(* IEC 61131-3 sources: std_i2980_v2.06_cp053/Source/IMM/ieccontrol/InjectionGeneral (part 3) *)

(* ---- ABBackPressureCalibCycle.pu ---- *)
(*
@h    ! WARNING !
@h    The Kemro K2 system (including software) only meets category B according to EN 954-1,
@h    thus it is not intended for usage in safety-relevant control applications in the field
@h    of personal safety (e.g. emergency stop).
@h    To implement potentially necessary safety-relevant control tasks, always use additional
@h    external safety devices that are intended for the particular purpose, and meet the necessary
@h    functional safety.
@h    For further information see EN 954-1 (EN ISO 13849-1) and/or the K2-x00 user manual, chapter
@h    "CE conformity, directives and standards".

Do steps for automatic hold pressure calibration
*)

IMPORT_OVER_LISTFILE
 SET_ALARM
, START_PROCESS_ALGORITHM
, cCompInjection
, cMoveFwd
, cMaxInjectionCount
, cMoveInjectCalib
, FBCheckReady
, tsDeviceId
, tevStartRequest
, tnOperationMode
, FBStopStartedMovements
, tsCalibMovement
, tsCalculatedInjectData2
, ABAutoCalibRedoListener
, tsControlParameters
, tsDeadTimeParameters
, tevStartRequestData
, tsCalculatedInjectData
, tyCalculatedDataArray
, tnCalibMode
, FBAutoCalibLog
, tsCalibShiftData
, KMEM_CreateData
, KMEM_Status

END_IMPORT

ALGORITHM_BLOCK ABBackPressureCalibCycle #DUMMY_EDIT_BLOCK

SYSTEM_VAR
 sv_OperationMode : tnOperationMode;
 sv_DeviceId : tsDeviceId;
 sv_CalibStateBackPressure : tsCalibMovement;
 sv_TmpInjectionData : tsCalculatedInjectData2;
 sv_bDoBackPressureCalib : BOOL;
 sv_HoldingControlParams : tsControlParameters;
 sv_HoldingDeadTimeParams : tsDeadTimeParameters;
END_VAR

SYSTEM_OBJECT
 TaskMid : TASK;
 evStartRequest : tevStartRequest;
 PU_Task_7 : TASK;
END_OBJECT

VAR
 fbCheckReady : FBCheckReady;
 InjDeviceId : tsDeviceId;
 fbStopStartedMovements : FBStopStartedMovements;
 abAutoCalibRedoListenerBackP : ABAutoCalibRedoListener;
END_VAR

PROCESS_ALGORITHM paRun ON TaskMid

VAR_TEMP
 tmpMeanData : tsCalculatedInjectData;
 i : DINT;
END_VAR

VAR
 evStartRequestData : tevStartRequestData;
 iInjectionCount : DINT;
 calculatedParameters : tyCalculatedDataArray;
 calibMode : tnCalibMode := tnCalibMode_Raising;
 fbLog : FBAutoCalibLog;
 ShiftData : tsCalibShiftData;
 ShiftArrayCreateData : KMEM_CreateData;
 MeasuredPresArrayCreateData : KMEM_CreateData;
 MeasuredOutputArrayCreateData : KMEM_CreateData;
 ThirdStageArrayCreateData : KMEM_CreateData;
 s : KMEM_Status;
 iSize : UDINT;
 rTmp : REAL;
END_VAR

(* IecGraph-Code *)

(* init step *)
INITIAL_STEP S_INIT:
AInit (P);
ACreateArrays (P);
END_STEP

ACTION AInit: #BEGIN_EDIT_BLOCK
InjDeviceId := sv_DeviceId;
sv_bDoBackPressureCalib := TRUE;
iInjectionCount := 1;
sv_TmpInjectionData.CalibMode := calibMode;
sv_TmpInjectionData.bValid := FALSE;

;#END_EDIT_BLOCK END_ACTION (*AInit*)

(* steps *)
STEP S_RESET:
AStopmovements (P);
Action24 (P);
END_STEP

ACTION Action24: #BEGIN_EDIT_BLOCK
IF sv_CalibStateBackPressure.Status <> tnCalibState_Error THEN
   sv_CalibStateBackPressure.Status := tnCalibState_Aborted;
   fbLog('Back pressure calib aborted');
ELSE
    fbLog('Back pressure calib error');
END_IF;

;#END_EDIT_BLOCK END_ACTION (*Action24*)
STEP S_STOP:
ADeleteArrays (P);
Action22 (P);
END_STEP

ACTION Action22: #BEGIN_EDIT_BLOCK
sv_bDoBackPressureCalib := FALSE;
STOP_PROCESS_ALGORITHM();

;#END_EDIT_BLOCK END_ACTION (*Action22*)
STEP S_INJECT:
ADoProfile (P);
Action9 (N);
END_STEP

ACTION Action9: #BEGIN_EDIT_BLOCK
fbCheckReady(DeviceId := InjDeviceId)

;#END_EDIT_BLOCK END_ACTION (*Action9*)
STEP S_WAIT_CALC:
END_STEP

STEP S_SAVE_CALC:
Action17 (P);
END_STEP

ACTION Action17: #BEGIN_EDIT_BLOCK
calculatedParameters[iInjectionCount] := sv_TmpInjectionData;

;#END_EDIT_BLOCK END_ACTION (*Action17*)
STEP S_NEXT_CYCLE:
Action16 (P);
END_STEP

ACTION Action16: #BEGIN_EDIT_BLOCK
iInjectionCount := iInjectionCount +1;

;#END_EDIT_BLOCK END_ACTION (*Action16*)
STEP S_DONE:
Action18 (P);
Action14 (P);
END_STEP

ACTION Action18: #BEGIN_EDIT_BLOCK
tmpMeanData.rControllerKR := 0.0;
tmpMeanData.rControllerW  := 0.0;
tmpMeanData.tPlantDeadTime:= t#0ms;
tmpMeanData.rPlantK       := 0.0;
tmpMeanData.tPlantT1      := t#0ms;
(* calculate mean value of all parameters *)
(* fixme: check if we need to calculate from falling and raising first
   and then calculate over the arry *)
FOR i:= 1 TO cMaxInjectionCount DO
    IF calibMode = tnCalibMode_Both THEN
        tmpMeanData.rControllerKR := tmpMeanData.rControllerKR + calculatedParameters[i].Falling.rControllerKR + calculatedParameters[i].Raising.rControllerKR;
        tmpMeanData.rControllerW  := tmpMeanData.rControllerW  + calculatedParameters[i].Falling.rControllerW  + calculatedParameters[i].Raising.rControllerW;
        tmpMeanData.tControllerTN := tmpMeanData.tControllerTN + calculatedParameters[i].Falling.tControllerTN + calculatedParameters[i].Raising.tControllerTN;
        tmpMeanData.tPlantDeadTime:= tmpMeanData.tPlantDeadTime+ calculatedParameters[i].Falling.tPlantDeadTime+ calculatedParameters[i].Raising.tPlantDeadTime;
        tmpMeanData.rPlantK       := tmpMeanData.rPlantK       + calculatedParameters[i].Falling.rPlantK       + calculatedParameters[i].Raising.rPlantK;
        tmpMeanData.tPlantT1      := tmpMeanData.tPlantT1      + calculatedParameters[i].Falling.tPlantT1      + calculatedParameters[i].Raising.tPlantT1;
       ELSIF calibMode = tnCalibMode_Raising THEN
        tmpMeanData.rControllerKR := tmpMeanData.rControllerKR + calculatedParameters[i].Raising.rControllerKR;
        tmpMeanData.rControllerW  := tmpMeanData.rControllerW  + calculatedParameters[i].Raising.rControllerW;
        tmpMeanData.tControllerTN := tmpMeanData.tControllerTN + calculatedParameters[i].Raising.tControllerTN;
        tmpMeanData.tPlantDeadTime:= tmpMeanData.tPlantDeadTime+ calculatedParameters[i].Raising.tPlantDeadTime;
        tmpMeanData.rPlantK       := tmpMeanData.rPlantK       + calculatedParameters[i].Raising.rPlantK;
        tmpMeanData.tPlantT1      := tmpMeanData.tPlantT1      + calculatedParameters[i].Raising.tPlantT1;
       ELSIF calibMode = tnCalibMode_Falling THEN
        tmpMeanData.rControllerKR := tmpMeanData.rControllerKR + calculatedParameters[i].Falling.rControllerKR ;
        tmpMeanData.rControllerW  := tmpMeanData.rControllerW  + calculatedParameters[i].Falling.rControllerW;
        tmpMeanData.tControllerTN := tmpMeanData.tControllerTN + calculatedParameters[i].Falling.tControllerTN;
        tmpMeanData.tPlantDeadTime:= tmpMeanData.tPlantDeadTime+ calculatedParameters[i].Falling.tPlantDeadTime;
        tmpMeanData.rPlantK       := tmpMeanData.rPlantK       + calculatedParameters[i].Falling.rPlantK;
        tmpMeanData.tPlantT1      := tmpMeanData.tPlantT1      + calculatedParameters[i].Falling.tPlantT1;
    END_IF;
END_FOR;

tmpMeanData.rControllerKR := tmpMeanData.rControllerKR / DINT_TO_REAL(cMaxInjectionCount);
tmpMeanData.rControllerW  := tmpMeanData.rControllerW  / DINT_TO_REAL(cMaxInjectionCount);
tmpMeanData.tControllerTN := tmpMeanData.tControllerTN / DINT_TO_REAL(cMaxInjectionCount);
tmpMeanData.tPlantDeadTime:= tmpMeanData.tPlantDeadTime/ DINT_TO_REAL(cMaxInjectionCount);
tmpMeanData.rPlantK       := tmpMeanData.rPlantK       / DINT_TO_REAL(cMaxInjectionCount);
tmpMeanData.tPlantT1      := tmpMeanData.tPlantT1      / DINT_TO_REAL(cMaxInjectionCount);

IF calibMode = tnCalibMode_Both THEN
    (* if only one edge no division is needed *)
    tmpMeanData.rControllerKR := tmpMeanData.rControllerKR / 2.0;
    tmpMeanData.rControllerW  := tmpMeanData.rControllerW  / 2.0;
    tmpMeanData.tControllerTN := DIVTIME(tmpMeanData.tControllerTN, 2);
    tmpMeanData.tPlantDeadTime:= DIVTIME(tmpMeanData.tPlantDeadTime, 2);
    tmpMeanData.rPlantK       := tmpMeanData.rPlantK/ 2.0;
    tmpMeanData.tPlantT1      := DIVTIME(tmpMeanData.tPlantT1, 2);
END_IF;

sv_HoldingControlParams.bUsePIDControl := TRUE;
sv_HoldingControlParams.rKS := 1.0;
sv_HoldingControlParams.dTN := tmpMeanData.tControllerTN;
sv_HoldingControlParams.dTV := t#0s;
sv_HoldingControlParams.rP := tmpMeanData.rControllerKR;

sv_HoldingDeadTimeParams.bCompensationEnabled := TRUE;
sv_HoldingDeadTimeParams.dDeadTime := tmpMeanData.tPlantDeadTime;
sv_HoldingDeadTimeParams.dPT2T1 := tmpMeanData.tPlantT1;
sv_HoldingDeadTimeParams.rPT2K := tmpMeanData.rPlantK;

sv_HoldingControlParams.bUsePIDControl := TRUE;

;#END_EDIT_BLOCK END_ACTION (*Action18*)
ACTION Action14: #BEGIN_EDIT_BLOCK
sv_CalibStateBackPressure.Status := tnCalibState_Done;

;#END_EDIT_BLOCK END_ACTION (*Action14*)

(* transitions *)
GO_ON_TRANSITION Trans15 (* Trans15 *) FROM S_RESET TO S_STOP :=  #BEGIN_EDIT_BLOCK
TRUE
;#END_EDIT_BLOCK
END_TRANSITION

TRANSITION Trans18 (* Trans18 *) FROM S_STOP TO S_INIT :=  #BEGIN_EDIT_BLOCK
TRUE
;#END_EDIT_BLOCK
END_TRANSITION

TRANSITION Trans1 (* Trans1 *) FROM S_INIT TO S_INJECT :=  #BEGIN_EDIT_BLOCK
TRUE
;#END_EDIT_BLOCK
END_TRANSITION

TRANSITION Trans2 (* Trans2 *) FROM S_INJECT TO S_WAIT_CALC :=  #BEGIN_EDIT_BLOCK
fbCheckReady.bReady AND S_INJECT.T >= t#1s
;#END_EDIT_BLOCK
(*Comment :FIXME: delay because else we sometimes get a erDeviceActive on first movement*)
END_TRANSITION

TRANSITION Trans21 (* Trans21 *) FROM S_WAIT_CALC TO S_SAVE_CALC :=  #BEGIN_EDIT_BLOCK
sv_TmpInjectionData.bValid
;#END_EDIT_BLOCK
END_TRANSITION

TRANSITION Trans22 (* Trans22 *) FROM S_WAIT_CALC TO S_RESET :=  #BEGIN_EDIT_BLOCK
sv_TmpInjectionData.bInvalid
;#END_EDIT_BLOCK
END_TRANSITION

TRANSITION Trans10 (* Trans10 *) FROM S_SAVE_CALC TO S_DONE :=  #BEGIN_EDIT_BLOCK
iInjectionCount >= cMaxInjectionCount
;#END_EDIT_BLOCK
END_TRANSITION

TRANSITION Trans11 (* Trans11 *) FROM S_SAVE_CALC TO S_NEXT_CYCLE :=  #BEGIN_EDIT_BLOCK
iInjectionCount < cMaxInjectionCount
;#END_EDIT_BLOCK
END_TRANSITION

TRANSITION Trans14 (* Trans14 *) FROM S_NEXT_CYCLE TO S_INJECT :=  #BEGIN_EDIT_BLOCK
TRUE
;#END_EDIT_BLOCK
END_TRANSITION

TRANSITION Trans19 (* Trans19 *) FROM S_DONE TO S_STOP :=  #BEGIN_EDIT_BLOCK
TRUE
;#END_EDIT_BLOCK
END_TRANSITION

(* end IecGraph-Code *)
(* sfc-code *)

(* stand alone actions *)
ACTION ADoProfile: #BEGIN_EDIT_BLOCK
evStartRequestData.DeviceId := InjDeviceId;
evStartRequestData.MoveDir := cMoveFwd;
evStartRequestData.MoveId := cMoveInjectCalib;
SET_EVENT(evStartRequest, evStartRequestData);

;#END_EDIT_BLOCK END_ACTION (*ADoProfile*)
ACTION AStopmovements: #BEGIN_EDIT_BLOCK
fbStopStartedMovements();

;#END_EDIT_BLOCK END_ACTION (*AStopmovements*)
ACTION ACreateArrays: #BEGIN_EDIT_BLOCK
(**************************************** WARNING ********************************************
 *** The KEBA Kemro K2 System including software is not intended for safety control tasks! ***
 ***                       For further information see Comment tab!                        ***
 *********************************************************************************************)

//create dynamic arrays which are necessary for PID parameter detection
iSize := DINT_TO_UDINT(cMaxShiftData) + 1;
ShiftArrayCreateData := KMEM_ArrayCreate(cCalibShiftData, ShiftData, iSize);

iSize := DINT_TO_UDINT(cMaxRecordedData);
MeasuredPresArrayCreateData := KMEM_ArrayCreate(cCalibMeasuredPres, rTmp, iSize);
MeasuredOutputArrayCreateData := KMEM_ArrayCreate(cCalibMeasuredOutput, rTmp, iSize);
ThirdStageArrayCreateData := KMEM_ArrayCreate(cCalibThirdStage, rTmp, iSize);

;#END_EDIT_BLOCK END_ACTION (*ACreateArrays*)
ACTION ADeleteArrays: #BEGIN_EDIT_BLOCK
(**************************************** WARNING ********************************************
 *** The KEBA Kemro K2 System including software is not intended for safety control tasks! ***
 ***                       For further information see Comment tab!                        ***
 *********************************************************************************************)

s := KMEM_ArrayDelete(ShiftArrayCreateData.Handle);
s := KMEM_ArrayDelete(MeasuredPresArrayCreateData.Handle);
s := KMEM_ArrayDelete(MeasuredOutputArrayCreateData.Handle);
s := KMEM_ArrayDelete(ThirdStageArrayCreateData.Handle);

;#END_EDIT_BLOCK END_ACTION (*ADeleteArrays*)

(* exits *)

EXIT_TRANSITION E_NotSetupMode := #BEGIN_EDIT_BLOCK
(**************************************** WARNING ********************************************
 *** The KEBA Kemro K2 System including software is not intended for safety control tasks! ***
 ***                       For further information see Comment tab!                        ***
 *********************************************************************************************)

sv_OperationMode <> nSetup
;#END_EDIT_BLOCK
PRIORITY 1 WITH  INITIAL_STEP S_RESET: END_STEP
END_TRANSITION

EXIT_TRANSITION E_NotCalibratingAnymore := #BEGIN_EDIT_BLOCK
// abort calibration, when not in running state and not finished
sv_CalibStateBackPressure.Status <> tnCalibState_Running AND (S_INIT.X (*OR S_FORWARD.X*) OR S_INJECT.X OR S_WAIT_CALC.X)
;#END_EDIT_BLOCK
PRIORITY 1 WITH  INITIAL_STEP S_RESET: END_STEP
END_TRANSITION
(* end sfc-code *)

END_ALGORITHM

POSTUPDATE_ALGORITHM pStart ON PU_Task_7 WITH sv_CalibStateBackPressure.Status

#BEGIN_EDIT_BLOCK
(**************************************** WARNING ********************************************
 *** The KEBA Kemro K2 System including software is not intended for safety control tasks! ***
 ***                       For further information see Comment tab!                        ***
 *********************************************************************************************)

IF sv_OperationMode = nSetup THEN
   IF sv_CalibStateBackPressure.Status = tnCalibState_Running THEN
      START_PROCESS_ALGORITHM(paRun);
   END_IF;
END_IF;

;#END_EDIT_BLOCK END_ALGORITHM

END_ALGORITHM_BLOCK

#END_OF_IEC_PART

@Puma @IecEditor 6 97 @Pou 25
@@@BEG_Comment@@@
@h    ! WARNING !
@h    The Kemro K2 system (including software) only meets category B according to EN 954-1,
@h    thus it is not intended for usage in safety-relevant control applications in the field
@h    of personal safety (e.g. emergency stop).
@h    To implement potentially necessary safety-relevant control tasks, always use additional
@h    external safety devices that are intended for the particular purpose, and meet the necessary
@h    functional safety.
@h    For further information see EN 954-1 (EN ISO 13849-1) and/or the K2-x00 user manual, chapter
@h    "CE conformity, directives and standards".

Do steps for automatic hold pressure calibration
@@@END_Comment@@@

@BEG_Contents

@BEG_Func
@RT(17)FuncTreeContainer
2
@Var @RT(9)SET_ALARM @RT(0) @T @T @DERIVED 0 @F @RT(23)KEBA_STANDARD_PROCEDURE @F
@T
@BEG_Attrib
0 @RT(0) @RT(0)
@END_Attrib
1 1 @F @F @F @F

@Var @RT(23)START_PROCESS_ALGORITHM @RT(0) @T @T @DERIVED 0 @F @RT(23)KEBA_STANDARD_PROCEDURE @F
@T
@BEG_Attrib
0 @RT(0) @RT(0)
@END_Attrib
1 1 @F @F @F @F

@END_Func

@BEG_Const
@RT(18)ConstTreeContainer
4
@Var @RT(14)cCompInjection @RT(0) @T @F @DT @RT(4)DINT @RT(0) @T @T @BASIC 0 @F
@F @F
@T
@BEG_Attrib
0 @RT(3)104 @RT(19)Component Injection
@END_Attrib
1 1 @F @F @F @F

@Var @RT(8)cMoveFwd @RT(0) @T @F @DT @RT(4)DINT @RT(0) @T @T @BASIC 0 @F
@F @F
@T
@BEG_Attrib
0 @RT(2)12 @RT(16)movement forward
@END_Attrib
1 1 @F @F @F @F

@Var @RT(18)cMaxInjectionCount @RT(0) @T @F @DT @RT(4)DINT @RT(0) @T @T @BASIC 0 @F
@F @F
@T
@BEG_Attrib
0 @RT(1)3 @RT(41)how often to do injection for calibration
@END_Attrib
1 1 @F @F @F @F

@Var @RT(16)cMoveInjectCalib @RT(0) @T @F @DT @RT(4)DINT @RT(0) @T @T @BASIC 0 @F
@F @F
@T
@BEG_Attrib
0 @RT(2)70 @RT(48)calibration movement for servo inject controller
@END_Attrib
1 1 @F @F @F @F

@END_Const

@BEG_Export

@BEG_Kind
@ALGORITHM_BLOCK @RT(24)ABBackPressureCalibCycle @STRUCTURED_TEXT
@RT(0) @RT(0) @RT(0)
@END_Kind

@BEG_Dcl
@RT(16)DclTreeContainer
14
@Var @RT(7)TaskMid @RT(0) @T @T @RENAMED 0 @T @T @DT @RT(4)TASK @RT(0) @T @T @BASIC 0 @F
@F @F
@T
@BEG_Attrib
3 @RT(0) @RT(0) @RT(0)
@END_Attrib
1 7 @F @F @F @F

@Var @RT(12)fbCheckReady @RT(0) @T @T @DERIVED 0 @T @T @DT @RT(12)FBCheckReady @RT(0) @T @T @UNKNOWN 0 @F
@F @F
@T
@BEG_Attrib
3 @RT(0) @RT(0) @RT(0)
@END_Attrib
1 0 @F @F @F @F

@Var @RT(11)InjDeviceId @RT(0) @T @T @DERIVED 0 @T @T @DT @RT(10)tsDeviceId @RT(0) @T @T @UNKNOWN 0 @F
@F @F
@T
@BEG_Attrib
3 @RT(0) @RT(0) @RT(0)
@END_Attrib
1 0 @F @F @F @F

@Var @RT(14)evStartRequest @RT(0) @T @T @DERIVED 0 @T @T @DT @RT(15)tevStartRequest @RT(0) @T @T @UNKNOWN 0 @F
@F @F
@T
@BEG_Attrib
3 @RT(0) @RT(0) @RT(0)
@END_Attrib
1 7 @F @F @F @F

@Var @RT(9)PU_Task_7 @RT(0) @T @T @RENAMED 0 @T @T @DT @RT(4)TASK @RT(0) @T @T @BASIC 0 @F
@F @F
@T
@BEG_Attrib
3 @RT(0) @RT(0) @RT(0)
@END_Attrib
1 7 @F @F @F @F

@Var @RT(16)sv_OperationMode @RT(0) @T @T @DERIVED 0 @T @T @DT @RT(15)tnOperationMode @RT(0) @T @T @UNKNOWN 0 @F
@F @F
@T
@BEG_Attrib
3 @RT(0) @RT(0) @RT(0)
@END_Attrib
1 8 @F @F @F @F

@Var @RT(22)fbStopStartedMovements @RT(0) @T @T @DERIVED 0 @T @T @DT @RT(22)FBStopStartedMovements @RT(0) @T @T @UNKNOWN 0 @F
@F @F
@T
@BEG_Attrib
3 @RT(0) @RT(0) @RT(0)
@END_Attrib
1 0 @F @F @F @F

@Var @RT(11)sv_DeviceId @RT(0) @T @T @RENAMED 0 @T @T @DT @RT(10)tsDeviceId @RT(0) @T @T @UNKNOWN 0 @F
@F @F
@T
@BEG_Attrib
3 @RT(0) @RT(0) @RT(0)
@END_Attrib
1 8 @F @F @F @F

@Var @RT(25)sv_CalibStateBackPressure @RT(0) @T @T @RENAMED 0 @T @T @DT @RT(15)tsCalibMovement @RT(0) @T @T @UNKNOWN 0 @F
@F @F
@T
@BEG_Attrib
3 @RT(0) @RT(0) @RT(0)
@END_Attrib
1 8 @F @F @F @F

@Var @RT(19)sv_TmpInjectionData @RT(0) @T @T @DERIVED 0 @T @T @DT @RT(23)tsCalculatedInjectData2 @RT(0) @T @T @UNKNOWN 0 @F
@F @F
@T
@BEG_Attrib
3 @RT(0) @RT(0) @RT(0)
@END_Attrib
1 8 @F @F @F @F

@Var @RT(23)sv_bDoBackPressureCalib @RT(0) @T @T @RENAMED 0 @T @T @DT @RT(4)BOOL @RT(0) @T @T @BASIC 0 @F
@F @F
@T
@BEG_Attrib
3 @RT(0) @RT(0) @RT(0)
@END_Attrib
1 8 @F @F @F @F

@Var @RT(28)abAutoCalibRedoListenerBackP @RT(0) @T @T @DERIVED 0 @T @T @DT @RT(23)ABAutoCalibRedoListener @RT(0) @T @T @UNKNOWN 0 @F
@F @F
@T
@BEG_Attrib
3 @RT(0) @RT(0) @RT(0)
@END_Attrib
1 0 @F @F @F @F

@Var @RT(23)sv_HoldingControlParams @RT(0) @T @T @RENAMED 0 @T @T @DT @RT(19)tsControlParameters @RT(0) @T @T @UNKNOWN 0 @F
@F @F
@T
@BEG_Attrib
3 @RT(0) @RT(0) @RT(0)
@END_Attrib
1 8 @F @F @F @F

@Var @RT(24)sv_HoldingDeadTimeParams @RT(0) @T @T @RENAMED 0 @T @T @DT @RT(20)tsDeadTimeParameters @RT(0) @T @T @UNKNOWN 0 @F
@F @F
@T
@BEG_Attrib
3 @RT(0) @RT(0) @RT(0)
@END_Attrib
1 8 @F @F @F @F

@END_Dcl

@END_Export

@BEG_Body

2

@BEG_Export

@BEG_Algo
@PROCESS_ALGORITHM @RT(5)paRun @SEQUENTIAL_FLOW_CHART
@RT(0) @RT(0) @RT(7)TaskMid @F @F
@END_Algo

@BEG_Dcl
@RT(16)DclTreeContainer
15
@Var @RT(18)evStartRequestData @RT(0) @T @T @DERIVED 0 @T @T @DT @RT(19)tevStartRequestData @RT(0) @T @T @UNKNOWN 0 @F
@F @F
@T
@BEG_Attrib
3 @RT(0) @RT(0) @RT(0)
@END_Attrib
1 0 @F @F @F @F

@Var @RT(15)iInjectionCount @RT(0) @T @F @DT @RT(4)DINT @RT(0) @T @T @BASIC 0 @F
@F @F
@T
@BEG_Attrib
3 @RT(0) @RT(0) @RT(0)
@END_Attrib
1 0 @F @F @F @F

@Var @RT(11)tmpMeanData @RT(0) @T @T @DERIVED 0 @T @T @DT @RT(22)tsCalculatedInjectData @RT(0) @T @T @UNKNOWN 0 @F
@F @F
@T
@BEG_Attrib
3 @RT(0) @RT(0) @RT(0)
@END_Attrib
1 4 @F @F @F @F

@Var @RT(20)calculatedParameters @RT(0) @T @T @DERIVED 0 @T @T @DT @RT(21)tyCalculatedDataArray @RT(0) @T @T @UNKNOWN 0 @F
@F @F
@T
@BEG_Attrib
3 @RT(0) @RT(0) @RT(0)
@END_Attrib
1 0 @F @F @F @F

@Var @RT(1)i @RT(0) @T @F @DT @RT(4)DINT @RT(0) @T @T @BASIC 0 @F
@F @F
@T
@BEG_Attrib
3 @RT(0) @RT(0) @RT(0)
@END_Attrib
1 4 @F @F @F @F

@Var @RT(9)calibMode @RT(0) @T @T @DERIVED 0 @T @T @DT @RT(11)tnCalibMode @RT(0) @T @T @UNKNOWN 0 @F
@F @F
@T
@BEG_Attrib
3 @RT(19)tnCalibMode_Raising @RT(0) @RT(0)
@END_Attrib
1 0 @F @F @F @F

@Var @RT(5)fbLog @RT(0) @T @T @DERIVED 0 @T @T @DT @RT(14)FBAutoCalibLog @RT(0) @T @T @UNKNOWN 0 @F
@F @F
@T
@BEG_Attrib
3 @RT(0) @RT(0) @RT(0)
@END_Attrib
1 0 @F @F @F @F

@Var @RT(9)ShiftData @RT(0) @T @T @DERIVED 0 @T @T @DT @RT(16)tsCalibShiftData @RT(0) @T @T @UNKNOWN 0 @F
@F @F
@T
@BEG_Attrib
3 @RT(0) @RT(0) @RT(0)
@END_Attrib
1 0 @F @F @F @F

@Var @RT(20)ShiftArrayCreateData @RT(0) @T @T @DERIVED 0 @T @T @DT @RT(15)KMEM_CreateData @RT(0) @T @T @UNKNOWN 0 @F
@F @F
@T
@BEG_Attrib
3 @RT(0) @RT(0) @RT(0)
@END_Attrib
1 0 @F @F @F @F

@Var @RT(27)MeasuredPresArrayCreateData @RT(0) @T @T @DERIVED 0 @T @T @DT @RT(15)KMEM_CreateData @RT(0) @T @T @UNKNOWN 0 @F
@F @F
@T
@BEG_Attrib
3 @RT(0) @RT(0) @RT(0)
@END_Attrib
1 0 @F @F @F @F

@Var @RT(29)MeasuredOutputArrayCreateData @RT(0) @T @T @DERIVED 0 @T @T @DT @RT(15)KMEM_CreateData @RT(0) @T @T @UNKNOWN 0 @F
@F @F
@T
@BEG_Attrib
3 @RT(0) @RT(0) @RT(0)
@END_Attrib
1 0 @F @F @F @F

@Var @RT(25)ThirdStageArrayCreateData @RT(0) @T @T @DERIVED 0 @T @T @DT @RT(15)KMEM_CreateData @RT(0) @T @T @UNKNOWN 0 @F
@F @F
@T
@BEG_Attrib
3 @RT(0) @RT(0) @RT(0)
@END_Attrib
1 0 @F @F @F @F

@Var @RT(1)s @RT(0) @T @T @DERIVED 0 @T @T @DT @RT(11)KMEM_Status @RT(0) @T @T @UNKNOWN 0 @F
@F @F
@T
@BEG_Attrib
3 @RT(0) @RT(0) @RT(0)
@END_Attrib
1 0 @F @F @F @F

@Var @RT(5)iSize @RT(0) @T @F @DT @RT(5)UDINT @RT(0) @T @T @BASIC 0 @F
@F @F
@T
@BEG_Attrib
3 @RT(0) @RT(0) @RT(0)
@END_Attrib
1 0 @F @F @F @F

@Var @RT(4)rTmp @RT(0) @T @F @DT @RT(4)REAL @RT(0) @T @T @BASIC 0 @F
@F @F
@T
@BEG_Attrib
3 @RT(0) @RT(0) @RT(0)
@END_Attrib
1 0 @F @F @F @F

@END_Dcl

@END_Export

@BEG_Export

@BEG_Algo
@POSTUPDATE_ALGORITHM @RT(6)pStart @STRUCTURED_TEXT
@RT(0) @RT(32)sv_CalibStateBackPressure.Status @RT(9)PU_Task_7 @F @F
@END_Algo

@BEG_Dcl
@RT(16)DclTreeContainer
0
@END_Dcl

@END_Export

@BEG_SfcBody
26 17 23

@BEG_SfcData 2
@StepSeq @RT(4)sseq @F 15
@Step @RT(7)S_RESET @F @F @T @F @RT(0) @F
@AcbCont @RT(7)unnamed @F 2
@Acb @RT(14)AStopmovements @F @F @RT(1)P @RT(0) @F @F @T @F
@Acb @RT(8)Action24 @F @T @RT(1)P @RT(0) @F @F @T @TL(7)
IF sv_CalibStateBackPressure.Status <> tnCalibState_Error THEN
   sv_CalibStateBackPressure.Status := tnCalibState_Aborted;
   fbLog('Back pressure calib aborted');
ELSE
    fbLog('Back pressure calib error');
END_IF;

@F

@Trans @RT(7)Trans15 @F @T @F @F @T @F @TL(2)
TRUE

@RT(7)Trans15 @F
@Step @RT(6)S_STOP @F @F @T @F @RT(0) @F
@AcbCont @RT(7)unnamed @F 2
@Acb @RT(13)ADeleteArrays @F @F @RT(1)P @RT(0) @F @F @F @F
@Acb @RT(8)Action22 @F @T @RT(1)P @RT(0) @F @F @T @TL(3)
sv_bDoBackPressureCalib := FALSE;
STOP_PROCESS_ALGORITHM();

@F

@Trans @RT(7)Trans18 @F @T @F @F @T @T @TL(2)
TRUE

@RT(7)Trans18 @F
@Step @RT(6)S_INIT @F @T @F @F @RT(0) @F
@AcbCont @RT(7)unnamed @F 2
@Acb @RT(5)AInit @F @T @RT(1)P @RT(0) @F @F @T @TL(6)
InjDeviceId := sv_DeviceId;
sv_bDoBackPressureCalib := TRUE;
iInjectionCount := 1;
sv_TmpInjectionData.CalibMode := calibMode;
sv_TmpInjectionData.bValid := FALSE;

@F
@Acb @RT(13)ACreateArrays @F @F @RT(1)P @RT(0) @F @F @F @F

@Trans @RT(6)Trans1 @F @T @F @F @T @T @TL(2)
TRUE

@RT(6)Trans1 @F
@Step @RT(8)S_INJECT @F @F @T @F @RT(0) @F
@AcbCont @RT(7)unnamed @F 2
@Acb @RT(10)ADoProfile @F @F @RT(1)P @RT(0) @F @F @T @F
@Acb @RT(7)Action9 @F @T @RT(1)N @RT(0) @F @F @T @TL(2)
fbCheckReady(DeviceId := InjDeviceId)

@F

@Trans @RT(6)Trans2 @F @T @F @F @T @T @TL(2)
fbCheckReady.bReady AND S_INJECT.T >= t#1s

@RT(6)Trans2 @T @TL(1)
Comment :FIXME: delay because else we sometimes get a erDeviceActive on first movement

@Step @RT(11)S_WAIT_CALC @F @F @F @F @RT(0) @F
@AcbCont @RT(7)unnamed @F 0

@AltBranch @RT(3)alt @F 2
@TransSeq @RT(4)tseq @F 1
@Trans @RT(7)Trans21 @F @T @F @F @T @T @TL(2)
sv_TmpInjectionData.bValid

@RT(7)Trans21 @F

@TransSeq @RT(4)tseq @F 2
@Trans @RT(7)Trans22 @F @T @F @F @T @T @TL(2)
sv_TmpInjectionData.bInvalid

@RT(7)Trans22 @F
@Goto @RT(7)S_RESET @F @F

@Step @RT(11)S_SAVE_CALC @F @F @F @F @RT(0) @F
@AcbCont @RT(7)unnamed @F 1
@Acb @RT(8)Action17 @F @T @RT(1)P @RT(0) @F @F @T @TL(2)
calculatedParameters[iInjectionCount] := sv_TmpInjectionData;

@F

@AltBranch @RT(3)alt @F 2
@TransSeq @RT(4)tseq @F 1
@Trans @RT(7)Trans10 @F @T @F @F @T @T @TL(2)
iInjectionCount >= cMaxInjectionCount

@RT(7)Trans10 @F

@TransSeq @RT(4)tseq @F 4
@Trans @RT(7)Trans11 @F @T @F @F @T @T @TL(2)
iInjectionCount < cMaxInjectionCount

@RT(7)Trans11 @F
@Step @RT(12)S_NEXT_CYCLE @F @F @F @F @RT(0) @F
@AcbCont @RT(7)unnamed @F 1
@Acb @RT(8)Action16 @F @T @RT(1)P @RT(0) @F @F @T @TL(2)
iInjectionCount := iInjectionCount +1;

@F

@Trans @RT(7)Trans14 @F @T @F @F @T @T @TL(2)
TRUE

@RT(7)Trans14 @F
@Goto @RT(8)S_INJECT @F @F

@Step @RT(6)S_DONE @F @F @F @F @RT(0) @F
@AcbCont @RT(7)unnamed @F 2
@Acb @RT(8)Action18 @F @T @RT(1)P @RT(0) @F @F @T @TL(63)
tmpMeanData.rControllerKR := 0.0;
tmpMeanData.rControllerW  := 0.0;
tmpMeanData.tPlantDeadTime:= t#0ms;
tmpMeanData.rPlantK       := 0.0;
tmpMeanData.tPlantT1      := t#0ms;
(* calculate mean value of all parameters *)
(* fixme: check if we need to calculate from falling and raising first
   and then calculate over the arry *)
FOR i:= 1 TO cMaxInjectionCount DO
    IF calibMode = tnCalibMode_Both THEN
        tmpMeanData.rControllerKR := tmpMeanData.rControllerKR + calculatedParameters[i].Falling.rControllerKR + calculatedParameters[i].Raising.rControllerKR;
        tmpMeanData.rControllerW  := tmpMeanData.rControllerW  + calculatedParameters[i].Falling.rControllerW  + calculatedParameters[i].Raising.rControllerW;
        tmpMeanData.tControllerTN := tmpMeanData.tControllerTN + calculatedParameters[i].Falling.tControllerTN + calculatedParameters[i].Raising.tControllerTN;
        tmpMeanData.tPlantDeadTime:= tmpMeanData.tPlantDeadTime+ calculatedParameters[i].Falling.tPlantDeadTime+ calculatedParameters[i].Raising.tPlantDeadTime;
        tmpMeanData.rPlantK       := tmpMeanData.rPlantK       + calculatedParameters[i].Falling.rPlantK       + calculatedParameters[i].Raising.rPlantK;
        tmpMeanData.tPlantT1      := tmpMeanData.tPlantT1      + calculatedParameters[i].Falling.tPlantT1      + calculatedParameters[i].Raising.tPlantT1;
       ELSIF calibMode = tnCalibMode_Raising THEN
        tmpMeanData.rControllerKR := tmpMeanData.rControllerKR + calculatedParameters[i].Raising.rControllerKR;
        tmpMeanData.rControllerW  := tmpMeanData.rControllerW  + calculatedParameters[i].Raising.rControllerW;
        tmpMeanData.tControllerTN := tmpMeanData.tControllerTN + calculatedParameters[i].Raising.tControllerTN;
        tmpMeanData.tPlantDeadTime:= tmpMeanData.tPlantDeadTime+ calculatedParameters[i].Raising.tPlantDeadTime;
        tmpMeanData.rPlantK       := tmpMeanData.rPlantK       + calculatedParameters[i].Raising.rPlantK;
        tmpMeanData.tPlantT1      := tmpMeanData.tPlantT1      + calculatedParameters[i].Raising.tPlantT1;
       ELSIF calibMode = tnCalibMode_Falling THEN
        tmpMeanData.rControllerKR := tmpMeanData.rControllerKR + calculatedParameters[i].Falling.rControllerKR ;
        tmpMeanData.rControllerW  := tmpMeanData.rControllerW  + calculatedParameters[i].Falling.rControllerW;
        tmpMeanData.tControllerTN := tmpMeanData.tControllerTN + calculatedParameters[i].Falling.tControllerTN;
        tmpMeanData.tPlantDeadTime:= tmpMeanData.tPlantDeadTime+ calculatedParameters[i].Falling.tPlantDeadTime;
        tmpMeanData.rPlantK       := tmpMeanData.rPlantK       + calculatedParameters[i].Falling.rPlantK;
        tmpMeanData.tPlantT1      := tmpMeanData.tPlantT1      + calculatedParameters[i].Falling.tPlantT1;
    END_IF;
END_FOR;

tmpMeanData.rControllerKR := tmpMeanData.rControllerKR / DINT_TO_REAL(cMaxInjectionCount);
tmpMeanData.rControllerW  := tmpMeanData.rControllerW  / DINT_TO_REAL(cMaxInjectionCount);
tmpMeanData.tControllerTN := tmpMeanData.tControllerTN / DINT_TO_REAL(cMaxInjectionCount);
tmpMeanData.tPlantDeadTime:= tmpMeanData.tPlantDeadTime/ DINT_TO_REAL(cMaxInjectionCount);
tmpMeanData.rPlantK       := tmpMeanData.rPlantK       / DINT_TO_REAL(cMaxInjectionCount);
tmpMeanData.tPlantT1      := tmpMeanData.tPlantT1      / DINT_TO_REAL(cMaxInjectionCount);

IF calibMode = tnCalibMode_Both THEN
    (* if only one edge no division is needed *)
    tmpMeanData.rControllerKR := tmpMeanData.rControllerKR / 2.0;
    tmpMeanData.rControllerW  := tmpMeanData.rControllerW  / 2.0;
    tmpMeanData.tControllerTN := DIVTIME(tmpMeanData.tControllerTN, 2);
    tmpMeanData.tPlantDeadTime:= DIVTIME(tmpMeanData.tPlantDeadTime, 2);
    tmpMeanData.rPlantK       := tmpMeanData.rPlantK/ 2.0;
    tmpMeanData.tPlantT1      := DIVTIME(tmpMeanData.tPlantT1, 2);
END_IF;

sv_HoldingControlParams.bUsePIDControl := TRUE;
sv_HoldingControlParams.rKS := 1.0;
sv_HoldingControlParams.dTN := tmpMeanData.tControllerTN;
sv_HoldingControlParams.dTV := t#0s;
sv_HoldingControlParams.rP := tmpMeanData.rControllerKR;

sv_HoldingDeadTimeParams.bCompensationEnabled := TRUE;
sv_HoldingDeadTimeParams.dDeadTime := tmpMeanData.tPlantDeadTime;
sv_HoldingDeadTimeParams.dPT2T1 := tmpMeanData.tPlantT1;
sv_HoldingDeadTimeParams.rPT2K := tmpMeanData.rPlantK;

sv_HoldingControlParams.bUsePIDControl := TRUE;

@F
@Acb @RT(8)Action14 @F @T @RT(1)P @RT(0) @F @F @T @TL(2)
sv_CalibStateBackPressure.Status := tnCalibState_Done;

@F

@Trans @RT(7)Trans19 @F @T @F @F @T @T @TL(2)
TRUE

@RT(7)Trans19 @F
@Goto @RT(6)S_STOP @F @F
@END_SfcData
@SaActions 4
@SaText @RT(10)ADoProfile 1 @TL(5)
evStartRequestData.DeviceId := InjDeviceId;
evStartRequestData.MoveDir := cMoveFwd;
evStartRequestData.MoveId := cMoveInjectCalib;
SET_EVENT(evStartRequest, evStartRequestData);

@SaText @RT(14)AStopmovements 1 @TL(2)
fbStopStartedMovements();

@SaText @RT(13)ACreateArrays 1 @TL(14)
(**************************************** WARNING ********************************************
 *** The KEBA Kemro K2 System including software is not intended for safety control tasks! ***
 ***                       For further information see Comment tab!                        ***
 *********************************************************************************************)

//create dynamic arrays which are necessary for PID parameter detection
iSize := DINT_TO_UDINT(cMaxShiftData) + 1;
ShiftArrayCreateData := KMEM_ArrayCreate(cCalibShiftData, ShiftData, iSize);

iSize := DINT_TO_UDINT(cMaxRecordedData);
MeasuredPresArrayCreateData := KMEM_ArrayCreate(cCalibMeasuredPres, rTmp, iSize);
MeasuredOutputArrayCreateData := KMEM_ArrayCreate(cCalibMeasuredOutput, rTmp, iSize);
ThirdStageArrayCreateData := KMEM_ArrayCreate(cCalibThirdStage, rTmp, iSize);

@SaText @RT(13)ADeleteArrays 1 @TL(10)
(**************************************** WARNING ********************************************
 *** The KEBA Kemro K2 System including software is not intended for safety control tasks! ***
 ***                       For further information see Comment tab!                        ***
 *********************************************************************************************)

s := KMEM_ArrayDelete(ShiftArrayCreateData.Handle);
s := KMEM_ArrayDelete(MeasuredPresArrayCreateData.Handle);
s := KMEM_ArrayDelete(MeasuredOutputArrayCreateData.Handle);
s := KMEM_ArrayDelete(ThirdStageArrayCreateData.Handle);

@SaTrans 0
@SaExits 2
@SaExit @SaText @RT(14)E_NotSetupMode 1 @TL(7)
(**************************************** WARNING ********************************************
 *** The KEBA Kemro K2 System including software is not intended for safety control tasks! ***
 ***                       For further information see Comment tab!                        ***
 *********************************************************************************************)

sv_OperationMode <> nSetup

@RT(7)S_RESET @RT(1)1 @F @F @SaSfc @RT(14)E_NotSetupMode 5 @RT(5)DUMMY
@BEG_SfcData 2
@ExitSeq @RT(4)sseq @F 3
@Step @RT(6)Step12 @F @T @F @F @RT(0) @F
@AcbCont @RT(7)unnamed @F 1
@Acb @RT(8)Action20 @F @F @RT(1)N @RT(0) @F @F @T @F

@Trans @RT(7)Trans16 @F @T @T @F @T @T @TL(2)
(*inl.*)

@RT(7)Trans16 @F
@Goto @RT(9)unlabeled @F @F
@END_SfcData

@SaExit @SaText @RT(23)E_NotCalibratingAnymore 1 @TL(3)
// abort calibration, when not in running state and not finished
sv_CalibStateBackPressure.Status <> tnCalibState_Running AND (S_INIT.X (*OR S_FORWARD.X*) OR S_INJECT.X OR S_WAIT_CALC.X)

@RT(7)S_RESET @RT(1)1 @F @F @SaSfc @RT(23)E_NotCalibratingAnymore 5 @RT(5)DUMMY
@BEG_SfcData 2
@ExitSeq @RT(4)sseq @F 3
@Step @RT(6)Step16 @F @T @F @F @RT(0) @F
@AcbCont @RT(7)unnamed @F 1
@Acb @RT(8)Action28 @F @F @RT(1)N @RT(0) @F @F @T @F

@Trans @RT(7)Trans22 @F @T @T @F @T @T @TL(2)
(*inl.*)

@RT(7)Trans22 @F
@Goto @RT(9)unlabeled @F @F
@END_SfcData

@END_SfcBody

@@@BEG_Comment@@@
@TL(0)

@@@END_Comment@@@

@BEG_Body
@TL(12)
(**************************************** WARNING ********************************************
 *** The KEBA Kemro K2 System including software is not intended for safety control tasks! ***
 ***                       For further information see Comment tab!                        ***
 *********************************************************************************************)

IF sv_OperationMode = nSetup THEN
   IF sv_CalibStateBackPressure.Status = tnCalibState_Running THEN
      START_PROCESS_ALGORITHM(paRun);
   END_IF;
END_IF;

@END_Body

@@@BEG_Comment@@@
@TL(0)

@@@END_Comment@@@
@END_Body

@END_Contents

(* ---- ABButtonControl.pu ---- *)
IMPORT_OVER_LISTFILE
 IS_LINKED
, tyPanelButton
, tevPanelButtonRegisterData
, tevPanelButtonRegister
, tsDeviceId
, ABManualButton
, tsPanelButton

END_IMPORT

ALGORITHM_BLOCK ABButtonControl #DUMMY_EDIT_BLOCK

SYSTEM_VAR
 sv_bInitStart : BOOL;
 sv_rScrewPosition : REAL;
 sv_bPlastEndReached : BOOL;
 sv_bInjectEnd : BOOL;
 sv_rScrewVolume : REAL;
 sv_iPanelMovementSelector : DINT;
 sv_PanelButtons : tyPanelButton;
 sv_DeviceId : tsDeviceId;
 sv_bDeviceReady : BOOL;
 di_ButtonInject : BOOL;
 di_ButtonDecomp : BOOL;
 di_ButtonPlast : BOOL;
 di_ButtonGeneral1 : BOOL;
 di_ButtonGeneral2 : BOOL;
 sv_bButtonInject : BOOL;
 sv_bButtonDecomp : BOOL;
 sv_bButtonPlast : BOOL;
END_VAR

SYSTEM_OBJECT
 evPanelButtonRegister : tevPanelButtonRegister;
 PU_Task_7 : TASK;
 PU_Task_13 : TASK;
END_OBJECT

VAR
 evPanelButtonRegisterData : tevPanelButtonRegisterData;
 abManualButton : ABManualButton;
 mpbButtonGeneralInject : REFTO BOOL;
 mpbButtonGeneralDecomp : REFTO BOOL;
 mpbButtonGeneralPlast : REFTO BOOL;
 mbDIButtonInjectLinked : BOOL;
 mbDIButtonPlastLinked : BOOL;
 mbDIButtonDecompLinked : BOOL;
 mbDIButtonGeneral1Linked : BOOL;
 mbDIButtonGeneral2Linked : BOOL;
 mpiPanelMovementSelector : REFTO DINT;
END_VAR

VAR CONSTANT
 cButtonMoveInjectDecomp : DINT := 1;
 cButtonMovePlast : DINT := 2;
END_VAR

POSTUPDATE_ALGORITHM pRegisterButtons ON PU_Task_13 WITH sv_bInitStart

#BEGIN_EDIT_BLOCK
(**************************************** WARNING ********************************************
 *** The KEBA Kemro K2 System including software is not intended for safety control tasks! ***
 ***                       For further information see Comment tab!                        ***
 *********************************************************************************************)

mpbButtonGeneralInject := EMPTY;
mpbButtonGeneralDecomp := EMPTY;
mpbButtonGeneralPlast := EMPTY;

mbDIButtonInjectLinked := IS_LINKED(di_ButtonInject);
mbDIButtonPlastLinked := IS_LINKED(di_ButtonPlast);
mbDIButtonDecompLinked := IS_LINKED(di_ButtonDecomp);

mbDIButtonGeneral1Linked := IS_LINKED(di_ButtonGeneral1);
mbDIButtonGeneral2Linked := IS_LINKED(di_ButtonGeneral2);

IF (mbDIButtonGeneral1Linked AND mbDIButtonGeneral2Linked) THEN
    mpiPanelMovementSelector := @sv_iPanelMovementSelector;
END_IF;

// register combined decomp-inject button
evPanelButtonRegisterData.Button.nPanelButtonType := nPanelButtonMovement;
evPanelButtonRegisterData.Button.iCompId := sv_DeviceId.CompId;
evPanelButtonRegisterData.Button.iIndexId := sv_DeviceId.IndexId;
evPanelButtonRegisterData.Button.iButtonId := cButtonMoveInjectDecomp;
evPanelButtonRegisterData.Button.pbActionVar1 := @sv_bButtonInject;
evPanelButtonRegisterData.Button.pbActionVar2 := @sv_bButtonDecomp;
evPanelButtonRegisterData.Button.Optional.pbLimitSwitch1 := @sv_bInjectEnd;
evPanelButtonRegisterData.Button.Optional.pbLimitSwitch2 := @sv_bPlastEndReached;
evPanelButtonRegisterData.Button.Optional.prActVar := @sv_rScrewPosition;
evPanelButtonRegisterData.Button.Optional.prMaxVar := @sv_rScrewVolume;
evPanelButtonRegisterData.Button.Optional.prMinVar :=  EMPTY;
evPanelButtonRegisterData.Button.Optional.iBarAttr := cBarInvert;
SET_EVENT(evPanelButtonRegister, evPanelButtonRegisterData);

// register plast button
evPanelButtonRegisterData.Button.nPanelButtonType := nPanelButtonMovement;
evPanelButtonRegisterData.Button.iCompId := sv_DeviceId.CompId;
evPanelButtonRegisterData.Button.iIndexId := sv_DeviceId.IndexId;
evPanelButtonRegisterData.Button.iButtonId := cButtonMovePlast;
evPanelButtonRegisterData.Button.pbActionVar1 := @sv_bButtonPlast;
evPanelButtonRegisterData.Button.pbActionVar2 := @sv_bButtonPlast;
evPanelButtonRegisterData.Button.Optional.pbLimitSwitch1 := EMPTY;
evPanelButtonRegisterData.Button.Optional.pbLimitSwitch2 := EMPTY;
evPanelButtonRegisterData.Button.Optional.prActVar := @sv_rScrewPosition;
evPanelButtonRegisterData.Button.Optional.prMaxVar := EMPTY;
evPanelButtonRegisterData.Button.Optional.prMinVar := EMPTY;
evPanelButtonRegisterData.Button.Optional.iBarAttr := 0;
SET_EVENT(evPanelButtonRegister, evPanelButtonRegisterData);

;#END_EDIT_BLOCK END_ALGORITHM

POSTUPDATE_ALGORITHM pButtonInject ON PU_Task_7 WITH di_ButtonInject, sv_bButtonInject,mpbButtonGeneralInject^

VAR
 bButton : BOOL;
END_VAR
#BEGIN_EDIT_BLOCK
(**************************************** WARNING ********************************************
 *** The KEBA Kemro K2 System including software is not intended for safety control tasks! ***
 ***                       For further information see Comment tab!                        ***
 *********************************************************************************************)

// soft panel button
bButton := sv_bButtonInject;

// hw panel button
IF mbDIButtonInjectLinked THEN
    bButton := bButton OR di_ButtonInject;
END_IF;

// external panel button
IF CHECK_REF(mpbButtonGeneralInject^) THEN
    bButton := bButton OR mpbButtonGeneralInject^;
END_IF;

abManualButton.aButtonInject(bButtonInject := bButton);

;#END_EDIT_BLOCK END_ALGORITHM

POSTUPDATE_ALGORITHM pButtonDecomp ON PU_Task_7 WITH di_ButtonDecomp, sv_bButtonDecomp,mpbButtonGeneralDecomp^

VAR
 bButton : BOOL;
END_VAR
#BEGIN_EDIT_BLOCK
(**************************************** WARNING ********************************************
 *** The KEBA Kemro K2 System including software is not intended for safety control tasks! ***
 ***                       For further information see Comment tab!                        ***
 *********************************************************************************************)

// soft panel button
bButton := sv_bButtonDecomp;

// hw panel button
IF mbDIButtonDecompLinked THEN
    bButton := bButton OR di_ButtonDecomp;
END_IF;

// external panel button
IF CHECK_REF(mpbButtonGeneralDecomp^) THEN
    bButton := bButton OR mpbButtonGeneralDecomp^;
END_IF;

abManualButton.aButtonDecomp(bButtonDecomp := bButton);

;#END_EDIT_BLOCK END_ALGORITHM

POSTUPDATE_ALGORITHM pButtonPlast ON PU_Task_7 WITH di_ButtonPlast, sv_bButtonPlast, mpbButtonGeneralPlast^

VAR
 bButton : BOOL;
END_VAR
#BEGIN_EDIT_BLOCK
(**************************************** WARNING ********************************************
 *** The KEBA Kemro K2 System including software is not intended for safety control tasks! ***
 ***                       For further information see Comment tab!                        ***
 *********************************************************************************************)

// soft panel button
bButton := sv_bButtonPlast;

// hw panel button
IF mbDIButtonPlastLinked THEN
    bButton := bButton OR di_ButtonPlast;
END_IF;

// external panel button
IF CHECK_REF(mpbButtonGeneralPlast^) THEN
    bButton := bButton OR mpbButtonGeneralPlast^;
END_IF;

abManualButton.aButtonPlast(bButtonPlast := bButton);

;#END_EDIT_BLOCK END_ALGORITHM

POSTUPDATE_ALGORITHM pMoveSelectorChanged ON PU_Task_7 WITH mpiPanelMovementSelector^

VAR
 Button : tsPanelButton;
END_VAR
#BEGIN_EDIT_BLOCK
(**************************************** WARNING ********************************************
 *** The KEBA Kemro K2 System including software is not intended for safety control tasks! ***
 ***                       For further information see Comment tab!                        ***
 *********************************************************************************************)

mpbButtonGeneralInject := EMPTY;
mpbButtonGeneralDecomp := EMPTY;
mpbButtonGeneralPlast := EMPTY;

IF (NOT sv_bDeviceReady) THEN
    // stop active movements
    abManualButton.aButtonInject(bButtonInject := FALSE);
    abManualButton.aButtonDecomp(bButtonDecomp := FALSE);
    abManualButton.aButtonPlast(bButtonPlast := FALSE);
END_IF;

IF (sv_iPanelMovementSelector > 0) THEN
    Button := sv_PanelButtons[sv_iPanelMovementSelector];
    IF (Button.iCompId = sv_DeviceId.CompId AND
        Button.iIndexId = sv_DeviceId.IndexId) THEN
        IF Button.iButtonId = cButtonMoveInjectDecomp THEN
            // combined inject/decomp
            mpbButtonGeneralInject := @di_ButtonGeneral1;
            mpbButtonGeneralDecomp := @di_ButtonGeneral2;
        ELSIF Button.iButtonId = cButtonMovePlast THEN
            // plast
            mpbButtonGeneralPlast := @di_ButtonGeneral1;
        END_IF;
    END_IF;
END_IF;

;#END_EDIT_BLOCK END_ALGORITHM

END_ALGORITHM_BLOCK

#END_OF_IEC_PART

@Puma @IecEditor 6 150 @Pou 25
@@@BEG_Comment@@@

@@@END_Comment@@@

@BEG_Contents

@BEG_Func
@RT(17)FuncTreeContainer
1
@Var @RT(9)IS_LINKED @RT(0) @T @T @DERIVED 0 @F @RT(22)KEBA_STANDARD_FUNCTION @F
@T
@BEG_Attrib
0 @RT(0) @RT(0)
@END_Attrib
1 1 @F @F @F @F

@END_Func

@BEG_Const
@RT(18)ConstTreeContainer
0
@END_Const

@BEG_Export

@BEG_Kind
@ALGORITHM_BLOCK @RT(15)ABButtonControl @STRUCTURED_TEXT
@RT(0) @RT(0) @RT(0)
@END_Kind

@BEG_Dcl
@RT(16)DclTreeContainer
33
@Var @RT(13)sv_bInitStart @RT(0) @T @T @RENAMED 0 @T @T @DT @RT(4)BOOL @RT(0) @T @T @BASIC 0 @F
@F @F
@T
@BEG_Attrib
3 @RT(0) @RT(0) @RT(0)
@END_Attrib
1 8 @F @F @F @F

@Var @RT(17)sv_rScrewPosition @RT(0) @T @F @DT @RT(4)REAL @RT(0) @T @T @BASIC 0 @F
@F @F
@T
@BEG_Attrib
3 @RT(0) @RT(0) @RT(0)
@END_Attrib
1 8 @F @F @F @F

@Var @RT(19)sv_bPlastEndReached @RT(0) @T @F @DT @RT(4)BOOL @RT(0) @T @T @BASIC 0 @F
@F @F
@T
@BEG_Attrib
3 @RT(0) @RT(0) @RT(0)
@END_Attrib
1 8 @F @F @F @F

@Var @RT(13)sv_bInjectEnd @RT(0) @T @F @DT @RT(4)BOOL @RT(0) @T @T @BASIC 0 @F
@F @F
@T
@BEG_Attrib
3 @RT(0) @RT(0) @RT(0)
@END_Attrib
1 8 @F @F @F @F

@Var @RT(15)sv_rScrewVolume @RT(0) @T @F @DT @RT(4)REAL @RT(0) @T @T @BASIC 0 @F
@F @F
@T
@BEG_Attrib
3 @RT(0) @RT(0) @RT(0)
@END_Attrib
1 8 @F @F @F @F

@Var @RT(25)sv_iPanelMovementSelector @RT(0) @T @F @DT @RT(4)DINT @RT(0) @T @T @BASIC 0 @F
@F @F
@T
@BEG_Attrib
3 @RT(0) @RT(0) @RT(0)
@END_Attrib
1 8 @F @F @F @F

@Var @RT(15)sv_PanelButtons @RT(0) @T @T @DERIVED 0 @T @T @DT @RT(13)tyPanelButton @RT(0) @T @T @UNKNOWN 0 @F
@F @F
@T
@BEG_Attrib
3 @RT(0) @RT(0) @RT(0)
@END_Attrib
1 8 @F @F @F @F

@Var @RT(25)evPanelButtonRegisterData @RT(0) @T @T @DERIVED 0 @T @T @DT @RT(26)tevPanelButtonRegisterData @RT(0) @T @T @UNKNOWN 0 @F
@F @F
@T
@BEG_Attrib
3 @RT(0) @RT(0) @RT(0)
@END_Attrib
1 0 @F @F @F @F

@Var @RT(21)evPanelButtonRegister @RT(0) @T @T @DERIVED 0 @T @T @DT @RT(22)tevPanelButtonRegister @RT(0) @T @T @UNKNOWN 0 @F
@F @F
@T
@BEG_Attrib
3 @RT(0) @RT(0) @RT(0)
@END_Attrib
1 7 @F @F @F @F

@Var @RT(11)sv_DeviceId @RT(0) @T @T @DERIVED 0 @T @T @DT @RT(10)tsDeviceId @RT(0) @T @T @UNKNOWN 0 @F
@F @F
@T
@BEG_Attrib
3 @RT(0) @RT(0) @RT(0)
@END_Attrib
1 8 @F @F @F @F

@Var @RT(15)sv_bDeviceReady @RT(0) @T @F @DT @RT(4)BOOL @RT(0) @T @T @BASIC 0 @F
@F @F
@T
@BEG_Attrib
3 @RT(0) @RT(0) @RT(0)
@END_Attrib
1 8 @F @F @F @F

@Var @RT(15)di_ButtonInject @RT(0) @T @T @RENAMED 0 @T @T @DT @RT(4)BOOL @RT(0) @T @T @BASIC 0 @F
@F @F
@T
@BEG_Attrib
3 @RT(0) @RT(0) @RT(0)
@END_Attrib
1 8 @F @F @F @F

@Var @RT(15)di_ButtonDecomp @RT(0) @T @T @RENAMED 0 @T @T @DT @RT(4)BOOL @RT(0) @T @T @BASIC 0 @F
@F @F
@T
@BEG_Attrib
3 @RT(0) @RT(0) @RT(0)
@END_Attrib
1 8 @F @F @F @F

@Var @RT(14)di_ButtonPlast @RT(0) @T @T @RENAMED 0 @T @T @DT @RT(4)BOOL @RT(0) @T @T @BASIC 0 @F
@F @F
@T
@BEG_Attrib
3 @RT(0) @RT(0) @RT(0)
@END_Attrib
1 8 @F @F @F @F

@Var @RT(17)di_ButtonGeneral1 @RT(0) @T @F @DT @RT(4)BOOL @RT(0) @T @T @BASIC 0 @F
@F @F
@T
@BEG_Attrib
3 @RT(0) @RT(0) @RT(0)
@END_Attrib
1 8 @F @F @F @F

@Var @RT(17)di_ButtonGeneral2 @RT(0) @T @F @DT @RT(4)BOOL @RT(0) @T @T @BASIC 0 @F
@F @F
@T
@BEG_Attrib
3 @RT(0) @RT(0) @RT(0)
@END_Attrib
1 8 @F @F @F @F

@Var @RT(16)sv_bButtonInject @RT(0) @T @F @DT @RT(4)BOOL @RT(0) @T @T @BASIC 0 @F
@F @F
@T
@BEG_Attrib
3 @RT(0) @RT(0) @RT(0)
@END_Attrib
1 8 @F @F @F @F

@Var @RT(16)sv_bButtonDecomp @RT(0) @T @F @DT @RT(4)BOOL @RT(0) @T @T @BASIC 0 @F
@F @F
@T
@BEG_Attrib
3 @RT(0) @RT(0) @RT(0)
@END_Attrib
1 8 @F @F @F @F

@Var @RT(15)sv_bButtonPlast @RT(0) @T @F @DT @RT(4)BOOL @RT(0) @T @T @BASIC 0 @F
@F @F
@T
@BEG_Attrib
3 @RT(0) @RT(0) @RT(0)
@END_Attrib
1 8 @F @F @F @F

@Var @RT(14)abManualButton @RT(0) @T @T @DERIVED 0 @T @T @DT @RT(14)ABManualButton @RT(0) @T @T @UNKNOWN 0 @F
@F @F
@T
@BEG_Attrib
3 @RT(0) @RT(0) @RT(0)
@END_Attrib
1 0 @F @F @F @F

@Var @RT(9)PU_Task_7 @RT(0) @T @F @DT @RT(4)TASK @RT(0) @T @T @BASIC 0 @F
@F @F
@T
@BEG_Attrib
3 @RT(0) @RT(0) @RT(0)
@END_Attrib
1 7 @F @F @F @F

@Var @RT(22)mpbButtonGeneralInject @RT(0) @T @T @REFTO 0 @T @DT @RT(4)BOOL @RT(0) @T @T @BASIC 0 @F
@F @F
@T
@BEG_Attrib
3 @RT(0) @RT(0) @RT(0)
@END_Attrib
1 0 @F @F @F @F

@Var @RT(22)mpbButtonGeneralDecomp @RT(0) @T @T @REFTO 0 @T @DT @RT(4)BOOL @RT(0) @T @T @BASIC 0 @F
@F @F
@T
@BEG_Attrib
3 @RT(0) @RT(0) @RT(0)
@END_Attrib
1 0 @F @F @F @F

@Var @RT(21)mpbButtonGeneralPlast @RT(0) @T @T @REFTO 0 @T @DT @RT(4)BOOL @RT(0) @T @T @BASIC 0 @F
@F @F
@T
@BEG_Attrib
3 @RT(0) @RT(0) @RT(0)
@END_Attrib
1 0 @F @F @F @F

@Var @RT(22)mbDIButtonInjectLinked @RT(0) @T @F @DT @RT(4)BOOL @RT(0) @T @T @BASIC 0 @F
@F @F
@T
@BEG_Attrib
3 @RT(0) @RT(0) @RT(0)
@END_Attrib
1 0 @F @F @F @F

@Var @RT(21)mbDIButtonPlastLinked @RT(0) @T @F @DT @RT(4)BOOL @RT(0) @T @T @BASIC 0 @F
@F @F
@T
@BEG_Attrib
3 @RT(0) @RT(0) @RT(0)
@END_Attrib
1 0 @F @F @F @F

@Var @RT(22)mbDIButtonDecompLinked @RT(0) @T @F @DT @RT(4)BOOL @RT(0) @T @T @BASIC 0 @F
@F @F
@T
@BEG_Attrib
3 @RT(0) @RT(0) @RT(0)
@END_Attrib
1 0 @F @F @F @F

@Var @RT(24)mbDIButtonGeneral1Linked @RT(0) @T @F @DT @RT(4)BOOL @RT(0) @T @T @BASIC 0 @F
@F @F
@T
@BEG_Attrib
3 @RT(0) @RT(0) @RT(0)
@END_Attrib
1 0 @F @F @F @F

@Var @RT(24)mbDIButtonGeneral2Linked @RT(0) @T @F @DT @RT(4)BOOL @RT(0) @T @T @BASIC 0 @F
@F @F
@T
@BEG_Attrib
3 @RT(0) @RT(0) @RT(0)
@END_Attrib
1 0 @F @F @F @F

@Var @RT(23)cButtonMoveInjectDecomp @RT(0) @T @F @DT @RT(4)DINT @RT(0) @T @T @BASIC 0 @F
@F @F
@T
@BEG_Attrib
3 @RT(1)1 @RT(0) @RT(0)
@END_Attrib
1 15 @F @F @F @F

@Var @RT(16)cButtonMovePlast @RT(0) @T @F @DT @RT(4)DINT @RT(0) @T @T @BASIC 0 @F
@F @F
@T
@BEG_Attrib
3 @RT(1)2 @RT(0) @RT(0)
@END_Attrib
1 15 @F @F @F @F

@Var @RT(10)PU_Task_13 @RT(0) @T @T @RENAMED 0 @T @T @DT @RT(4)TASK @RT(0) @T @T @BASIC 0 @F
@F @F
@T
@BEG_Attrib
3 @RT(0) @RT(0) @RT(0)
@END_Attrib
1 7 @F @F @F @F

@Var @RT(24)mpiPanelMovementSelector @RT(0) @T @T @REFTO 0 @T @DT @RT(4)DINT @RT(0) @T @T @BASIC 0 @F
@F @F
@T
@BEG_Attrib
3 @RT(0) @RT(0) @RT(0)
@END_Attrib
1 0 @F @F @F @F

@END_Dcl

@END_Export

@BEG_Body

5

@BEG_Export

@BEG_Algo
@POSTUPDATE_ALGORITHM @RT(16)pRegisterButtons @STRUCTURED_TEXT
@RT(0) @RT(13)sv_bInitStart @RT(10)PU_Task_13 @F @F
@END_Algo

@BEG_Dcl
@RT(16)DclTreeContainer
0
@END_Dcl

@END_Export

@BEG_Export

@BEG_Algo
@POSTUPDATE_ALGORITHM @RT(13)pButtonInject @STRUCTURED_TEXT
@RT(0) @RT(57)di_ButtonInject, sv_bButtonInject,mpbButtonGeneralInject^ @RT(9)PU_Task_7 @F @F
@END_Algo

@BEG_Dcl
@RT(16)DclTreeContainer
1
@Var @RT(7)bButton @RT(0) @T @F @DT @RT(4)BOOL @RT(0) @T @T @BASIC 0 @F
@F @F
@T
@BEG_Attrib
3 @RT(0) @RT(0) @RT(0)
@END_Attrib
1 0 @F @F @F @F

@END_Dcl

@END_Export

@BEG_Export

@BEG_Algo
@POSTUPDATE_ALGORITHM @RT(13)pButtonDecomp @STRUCTURED_TEXT
@RT(0) @RT(57)di_ButtonDecomp, sv_bButtonDecomp,mpbButtonGeneralDecomp^ @RT(9)PU_Task_7 @F @F
@END_Algo

@BEG_Dcl
@RT(16)DclTreeContainer
1
@Var @RT(7)bButton @RT(0) @T @F @DT @RT(4)BOOL @RT(0) @T @T @BASIC 0 @F
@F @F
@T
@BEG_Attrib
3 @RT(0) @RT(0) @RT(0)
@END_Attrib
1 0 @F @F @F @F

@END_Dcl

@END_Export

@BEG_Export

@BEG_Algo
@POSTUPDATE_ALGORITHM @RT(12)pButtonPlast @STRUCTURED_TEXT
@RT(0) @RT(55)di_ButtonPlast, sv_bButtonPlast, mpbButtonGeneralPlast^ @RT(9)PU_Task_7 @F @F
@END_Algo

@BEG_Dcl
@RT(16)DclTreeContainer
1
@Var @RT(7)bButton @RT(0) @T @F @DT @RT(4)BOOL @RT(0) @T @T @BASIC 0 @F
@F @F
@T
@BEG_Attrib
3 @RT(0) @RT(0) @RT(0)
@END_Attrib
1 0 @F @F @F @F

@END_Dcl

@END_Export

@BEG_Export

@BEG_Algo
@POSTUPDATE_ALGORITHM @RT(20)pMoveSelectorChanged @STRUCTURED_TEXT
@RT(0) @RT(25)mpiPanelMovementSelector^ @RT(9)PU_Task_7 @F @F
@END_Algo

@BEG_Dcl
@RT(16)DclTreeContainer
1
@Var @RT(6)Button @RT(0) @T @T @DERIVED 0 @T @T @DT @RT(13)tsPanelButton @RT(0) @T @T @UNKNOWN 0 @F
@F @F
@T
@BEG_Attrib
3 @RT(0) @RT(0) @RT(0)
@END_Attrib
1 0 @F @F @F @F

@END_Dcl

@END_Export

@BEG_Body
@TL(50)
(**************************************** WARNING ********************************************
 *** The KEBA Kemro K2 System including software is not intended for safety control tasks! ***
 ***                       For further information see Comment tab!                        ***
 *********************************************************************************************)

mpbButtonGeneralInject := EMPTY;
mpbButtonGeneralDecomp := EMPTY;
mpbButtonGeneralPlast := EMPTY;

mbDIButtonInjectLinked := IS_LINKED(di_ButtonInject);
mbDIButtonPlastLinked := IS_LINKED(di_ButtonPlast);
mbDIButtonDecompLinked := IS_LINKED(di_ButtonDecomp);

mbDIButtonGeneral1Linked := IS_LINKED(di_ButtonGeneral1);
mbDIButtonGeneral2Linked := IS_LINKED(di_ButtonGeneral2);

IF (mbDIButtonGeneral1Linked AND mbDIButtonGeneral2Linked) THEN
    mpiPanelMovementSelector := @sv_iPanelMovementSelector;
END_IF;

// register combined decomp-inject button
evPanelButtonRegisterData.Button.nPanelButtonType := nPanelButtonMovement;
evPanelButtonRegisterData.Button.iCompId := sv_DeviceId.CompId;
evPanelButtonRegisterData.Button.iIndexId := sv_DeviceId.IndexId;
evPanelButtonRegisterData.Button.iButtonId := cButtonMoveInjectDecomp;
evPanelButtonRegisterData.Button.pbActionVar1 := @sv_bButtonInject;
evPanelButtonRegisterData.Button.pbActionVar2 := @sv_bButtonDecomp;
evPanelButtonRegisterData.Button.Optional.pbLimitSwitch1 := @sv_bInjectEnd;
evPanelButtonRegisterData.Button.Optional.pbLimitSwitch2 := @sv_bPlastEndReached;
evPanelButtonRegisterData.Button.Optional.prActVar := @sv_rScrewPosition;
evPanelButtonRegisterData.Button.Optional.prMaxVar := @sv_rScrewVolume;
evPanelButtonRegisterData.Button.Optional.prMinVar :=  EMPTY;
evPanelButtonRegisterData.Button.Optional.iBarAttr := cBarInvert;
SET_EVENT(evPanelButtonRegister, evPanelButtonRegisterData);

// register plast button
evPanelButtonRegisterData.Button.nPanelButtonType := nPanelButtonMovement;
evPanelButtonRegisterData.Button.iCompId := sv_DeviceId.CompId;
evPanelButtonRegisterData.Button.iIndexId := sv_DeviceId.IndexId;
evPanelButtonRegisterData.Button.iButtonId := cButtonMovePlast;
evPanelButtonRegisterData.Button.pbActionVar1 := @sv_bButtonPlast;
evPanelButtonRegisterData.Button.pbActionVar2 := @sv_bButtonPlast;
evPanelButtonRegisterData.Button.Optional.pbLimitSwitch1 := EMPTY;
evPanelButtonRegisterData.Button.Optional.pbLimitSwitch2 := EMPTY;
evPanelButtonRegisterData.Button.Optional.prActVar := @sv_rScrewPosition;
evPanelButtonRegisterData.Button.Optional.prMaxVar := EMPTY;
evPanelButtonRegisterData.Button.Optional.prMinVar := EMPTY;
evPanelButtonRegisterData.Button.Optional.iBarAttr := 0;
SET_EVENT(evPanelButtonRegister, evPanelButtonRegisterData);

@END_Body

@@@BEG_Comment@@@
@TL(0)

@@@END_Comment@@@

@BEG_Body
@TL(20)
(**************************************** WARNING ********************************************
 *** The KEBA Kemro K2 System including software is not intended for safety control tasks! ***
 ***                       For further information see Comment tab!                        ***
 *********************************************************************************************)

// soft panel button
bButton := sv_bButtonInject;

// hw panel button
IF mbDIButtonInjectLinked THEN
    bButton := bButton OR di_ButtonInject;
END_IF;

// external panel button
IF CHECK_REF(mpbButtonGeneralInject^) THEN
    bButton := bButton OR mpbButtonGeneralInject^;
END_IF;

abManualButton.aButtonInject(bButtonInject := bButton);

@END_Body

@@@BEG_Comment@@@
@TL(0)

@@@END_Comment@@@

@BEG_Body
@TL(21)
(**************************************** WARNING ********************************************
 *** The KEBA Kemro K2 System including software is not intended for safety control tasks! ***
 ***                       For further information see Comment tab!                        ***
 *********************************************************************************************)

// soft panel button
bButton := sv_bButtonDecomp;

// hw panel button
IF mbDIButtonDecompLinked THEN
    bButton := bButton OR di_ButtonDecomp;
END_IF;

// external panel button
IF CHECK_REF(mpbButtonGeneralDecomp^) THEN
    bButton := bButton OR mpbButtonGeneralDecomp^;
END_IF;

abManualButton.aButtonDecomp(bButtonDecomp := bButton);

@END_Body

@@@BEG_Comment@@@
@TL(0)

@@@END_Comment@@@

@BEG_Body
@TL(21)
(**************************************** WARNING ********************************************
 *** The KEBA Kemro K2 System including software is not intended for safety control tasks! ***
 ***                       For further information see Comment tab!                        ***
 *********************************************************************************************)

// soft panel button
bButton := sv_bButtonPlast;

// hw panel button
IF mbDIButtonPlastLinked THEN
    bButton := bButton OR di_ButtonPlast;
END_IF;

// external panel button
IF CHECK_REF(mpbButtonGeneralPlast^) THEN
    bButton := bButton OR mpbButtonGeneralPlast^;
END_IF;

abManualButton.aButtonPlast(bButtonPlast := bButton);

@END_Body

@@@BEG_Comment@@@
@TL(0)

@@@END_Comment@@@

@BEG_Body
@TL(31)
(**************************************** WARNING ********************************************
 *** The KEBA Kemro K2 System including software is not intended for safety control tasks! ***
 ***                       For further information see Comment tab!                        ***
 *********************************************************************************************)

mpbButtonGeneralInject := EMPTY;
mpbButtonGeneralDecomp := EMPTY;
mpbButtonGeneralPlast := EMPTY;

IF (NOT sv_bDeviceReady) THEN
    // stop active movements
    abManualButton.aButtonInject(bButtonInject := FALSE);
    abManualButton.aButtonDecomp(bButtonDecomp := FALSE);
    abManualButton.aButtonPlast(bButtonPlast := FALSE);
END_IF;

IF (sv_iPanelMovementSelector > 0) THEN
    Button := sv_PanelButtons[sv_iPanelMovementSelector];
    IF (Button.iCompId = sv_DeviceId.CompId AND
        Button.iIndexId = sv_DeviceId.IndexId) THEN
        IF Button.iButtonId = cButtonMoveInjectDecomp THEN
            // combined inject/decomp
            mpbButtonGeneralInject := @di_ButtonGeneral1;
            mpbButtonGeneralDecomp := @di_ButtonGeneral2;
        ELSIF Button.iButtonId = cButtonMovePlast THEN
            // plast
            mpbButtonGeneralPlast := @di_ButtonGeneral1;
        END_IF;
    END_IF;
END_IF;

@END_Body

@@@BEG_Comment@@@
@TL(0)

@@@END_Comment@@@
@END_Body

@END_Contents

(* ---- ABChangeProfile.pu ---- *)
(*
@h    ! WARNING !
@h    The Kemro K2 system (including software) only meets category B according to EN 954-1,
@h    thus it is not intended for usage in safety-relevant control applications in the field
@h    of personal safety (e.g. emergency stop).
@h    To implement potentially necessary safety-relevant control tasks, always use additional
@h    external safety devices that are intended for the particular purpose, and meet the necessary
@h    functional safety.
@h    For further information see EN 954-1 (EN ISO 13849-1) and/or the K2-x00 user manual, chapter
@h    "CE conformity, directives and standards".

This AB includes the following functions:

+ reorder inject profile after number of inject profile stages changed
+ reorder plast profile after number of plast profile stages changed
+ copy screw volume to start position of first inject profile point after mold data loading
*)

IMPORT_OVER_LISTFILE
 KAPPL_VisProfilePlast
, KAPPL_VisProfile
, tnDataState
, FBChangeNoOfProfileSteps
, FBChangeNoOfProfileStepsPlast

END_IMPORT

ALGORITHM_BLOCK ABChangeProfile #DUMMY_EDIT_BLOCK

SYSTEM_VAR
 sv_bUseStartPosProfiles : BOOL;
 sv_PlastProfVis : KAPPL_VisProfilePlast;
 sv_bInitStart : BOOL;
 sv_InjectProfVis : KAPPL_VisProfile;
 sv_DataState : tnDataState;
 sv_rScrewVolume : REAL;
END_VAR

SYSTEM_OBJECT
 PU_Task_7 : TASK;
END_OBJECT

POSTUPDATE_ALGORITHM pChangeInjectProfile ON PU_Task_7 WITH sv_InjectProfVis, sv_bInitStart

VAR
 fbChangeNoOfProfileSteps : FBChangeNoOfProfileSteps;
END_VAR
#BEGIN_EDIT_BLOCK
fbChangeNoOfProfileSteps(ProfileVis := sv_InjectProfVis.Profile,
                         bUseStartPosProfiles := sv_bUseStartPosProfiles,
                         bOpenEndProfile := sv_InjectProfVis.bOpenEndProfile,
                         bDataStateIsReady := (sv_DataState = nReady));

;#END_EDIT_BLOCK END_ALGORITHM

POSTUPDATE_ALGORITHM pChangePlastProfile ON PU_Task_7 WITH sv_PlastProfVis,sv_bInitStart

VAR
 fbChangeNoOfProfileStepsPlast : FBChangeNoOfProfileStepsPlast;
END_VAR
#BEGIN_EDIT_BLOCK
fbChangeNoOfProfileStepsPlast(ProfileVis := sv_PlastProfVis.Profile,
                              bUseStartPosProfiles := sv_bUseStartPosProfiles,
                              bOpenEndProfile := sv_PlastProfVis.bOpenEndProfile,
                              bDataStateIsReady := (sv_DataState = nReady));

;#END_EDIT_BLOCK END_ALGORITHM

POSTUPDATE_ALGORITHM pNewMoldData ON PU_Task_7 WITH sv_DataState

VAR
 bLoadingInProgress : BOOL;
END_VAR
#BEGIN_EDIT_BLOCK
(**************************************** WARNING ********************************************
 *** The KEBA Kemro K2 System including software is not intended for safety control tasks! ***
 ***                       For further information see Comment tab!                        ***
 *********************************************************************************************)

IF sv_DataState = nReadMoldData THEN
   //loading of mold data in progress
   bLoadingInProgress := TRUE;
   RETURN;
END_IF;

IF sv_DataState = nReady AND bLoadingInProgress THEN

   //copy screw volume to first profile point of inject profile
   //(this profile point is not visible on hmi)
   sv_InjectProfVis.Profile.Points[1].rStartPos := sv_rScrewVolume;

   bLoadingInProgress := FALSE;

END_IF;

;#END_EDIT_BLOCK END_ALGORITHM

END_ALGORITHM_BLOCK

#END_OF_IEC_PART

@Puma @IecEditor 6 103 @Pou 25
@@@BEG_Comment@@@
@h    ! WARNING !
@h    The Kemro K2 system (including software) only meets category B according to EN 954-1,
@h    thus it is not intended for usage in safety-relevant control applications in the field
@h    of personal safety (e.g. emergency stop).
@h    To implement potentially necessary safety-relevant control tasks, always use additional
@h    external safety devices that are intended for the particular purpose, and meet the necessary
@h    functional safety.
@h    For further information see EN 954-1 (EN ISO 13849-1) and/or the K2-x00 user manual, chapter
@h    "CE conformity, directives and standards".

This AB includes the following functions:

+ reorder inject profile after number of inject profile stages changed
+ reorder plast profile after number of plast profile stages changed
+ copy screw volume to start position of first inject profile point after mold data loading
@@@END_Comment@@@

@BEG_Contents

@BEG_Func
@RT(17)FuncTreeContainer
0
@END_Func

@BEG_Const
@RT(18)ConstTreeContainer
0
@END_Const

@BEG_Export

@BEG_Kind
@ALGORITHM_BLOCK @RT(15)ABChangeProfile @STRUCTURED_TEXT
@RT(0) @RT(0) @RT(0)
@END_Kind

@BEG_Dcl
@RT(16)DclTreeContainer
7
@Var @RT(9)PU_Task_7 @RT(0) @T @T @RENAMED 0 @T @T @DT @RT(4)TASK @RT(0) @T @T @BASIC 0 @F
@F @F
@T
@BEG_Attrib
3 @RT(0) @RT(0) @RT(0)
@END_Attrib
1 7 @F @F @F @F

@Var @RT(23)sv_bUseStartPosProfiles @RT(0) @T @F @DT @RT(4)BOOL @RT(0) @T @T @BASIC 0 @F
@F @F
@T
@BEG_Attrib
3 @RT(0) @RT(0) @RT(0)
@END_Attrib
1 8 @F @F @F @F

@Var @RT(15)sv_PlastProfVis @RT(0) @T @T @DERIVED 0 @T @T @DT @RT(21)KAPPL_VisProfilePlast @RT(0) @T @T @UNKNOWN 0 @F
@F @F
@T
@BEG_Attrib
3 @RT(0) @RT(0) @RT(0)
@END_Attrib
1 8 @F @F @F @F

@Var @RT(13)sv_bInitStart @RT(0) @T @F @DT @RT(4)BOOL @RT(0) @T @T @BASIC 0 @F
@F @F
@T
@BEG_Attrib
3 @RT(0) @RT(0) @RT(0)
@END_Attrib
1 8 @F @F @F @F

@Var @RT(16)sv_InjectProfVis @RT(0) @T @T @DERIVED 0 @F @RT(16)KAPPL_VisProfile @F
@T
@BEG_Attrib
3 @RT(0) @RT(0) @RT(0)
@END_Attrib
1 8 @F @F @F @F

@Var @RT(12)sv_DataState @RT(0) @T @T @DERIVED 0 @T @T @DT @RT(11)tnDataState @RT(0) @T @T @UNKNOWN 0 @F
@F @F
@T
@BEG_Attrib
3 @RT(0) @RT(0) @RT(0)
@END_Attrib
1 8 @F @F @F @F

@Var @RT(15)sv_rScrewVolume @RT(0) @T @F @DT @RT(4)REAL @RT(0) @T @T @BASIC 0 @F
@F @F
@T
@BEG_Attrib
3 @RT(0) @RT(0) @RT(0)
@END_Attrib
1 8 @F @F @F @F

@END_Dcl

@END_Export

@BEG_Body

3

@BEG_Export

@BEG_Algo
@POSTUPDATE_ALGORITHM @RT(20)pChangeInjectProfile @STRUCTURED_TEXT
@RT(0) @RT(31)sv_InjectProfVis, sv_bInitStart @RT(9)PU_Task_7 @F @F
@END_Algo

@BEG_Dcl
@RT(16)DclTreeContainer
1
@Var @RT(24)fbChangeNoOfProfileSteps @RT(0) @T @T @DERIVED 0 @T @T @DT @RT(24)FBChangeNoOfProfileSteps @RT(0) @T @T @UNKNOWN 0 @F
@F @F
@T
@BEG_Attrib
3 @RT(0) @RT(0) @RT(0)
@END_Attrib
1 0 @F @F @F @F

@END_Dcl

@END_Export

@BEG_Export

@BEG_Algo
@POSTUPDATE_ALGORITHM @RT(19)pChangePlastProfile @STRUCTURED_TEXT
@RT(0) @RT(29)sv_PlastProfVis,sv_bInitStart @RT(9)PU_Task_7 @F @F
@END_Algo

@BEG_Dcl
@RT(16)DclTreeContainer
1
@Var @RT(29)fbChangeNoOfProfileStepsPlast @RT(0) @T @T @DERIVED 0 @T @T @DT @RT(29)FBChangeNoOfProfileStepsPlast @RT(0) @T @T @UNKNOWN 0 @F
@F @F
@T
@BEG_Attrib
3 @RT(0) @RT(0) @RT(0)
@END_Attrib
1 0 @F @F @F @F

@END_Dcl

@END_Export

@BEG_Export

@BEG_Algo
@POSTUPDATE_ALGORITHM @RT(12)pNewMoldData @STRUCTURED_TEXT
@RT(0) @RT(12)sv_DataState @RT(9)PU_Task_7 @F @F
@END_Algo

@BEG_Dcl
@RT(16)DclTreeContainer
1
@Var @RT(18)bLoadingInProgress @RT(0) @T @F @DT @RT(4)BOOL @RT(0) @T @T @BASIC 0 @F
@F @F
@T
@BEG_Attrib
3 @RT(0) @RT(0) @RT(0)
@END_Attrib
1 0 @F @F @F @F

@END_Dcl

@END_Export

@BEG_Body
@TL(6)
fbChangeNoOfProfileSteps(ProfileVis := sv_InjectProfVis.Profile,
                         bUseStartPosProfiles := sv_bUseStartPosProfiles,
                         bOpenEndProfile := sv_InjectProfVis.bOpenEndProfile,
                         bDataStateIsReady := (sv_DataState = nReady));

@END_Body

@@@BEG_Comment@@@
@TL(0)

@@@END_Comment@@@

@BEG_Body
@TL(6)
fbChangeNoOfProfileStepsPlast(ProfileVis := sv_PlastProfVis.Profile,
                              bUseStartPosProfiles := sv_bUseStartPosProfiles,
                              bOpenEndProfile := sv_PlastProfVis.bOpenEndProfile,
                              bDataStateIsReady := (sv_DataState = nReady));

@END_Body

@@@BEG_Comment@@@
@TL(0)

@@@END_Comment@@@

@BEG_Body
@TL(21)
(**************************************** WARNING ********************************************
 *** The KEBA Kemro K2 System including software is not intended for safety control tasks! ***
 ***                       For further information see Comment tab!                        ***
 *********************************************************************************************)

IF sv_DataState = nReadMoldData THEN
   //loading of mold data in progress
   bLoadingInProgress := TRUE;
   RETURN;
END_IF;

IF sv_DataState = nReady AND bLoadingInProgress THEN

   //copy screw volume to first profile point of inject profile
   //(this profile point is not visible on hmi)
   sv_InjectProfVis.Profile.Points[1].rStartPos := sv_rScrewVolume;

   bLoadingInProgress := FALSE;

END_IF;

@END_Body

@@@BEG_Comment@@@
@TL(0)

@@@END_Comment@@@
@END_Body

@END_Contents

(* ---- ABCheckColdDropPossible.pu ---- *)
(*
@h    ! WARNING !
@h    The Kemro K2 system (including software) only meets category B according to EN 954-1,
@h    thus it is not intended for usage in safety-relevant control applications in the field
@h    of personal safety (e.g. emergency stop).
@h    To implement potentially necessary safety-relevant control tasks, always use additional
@h    external safety devices that are intended for the particular purpose, and meet the necessary
@h    functional safety.
@h    For further information see EN 954-1 (EN ISO 13849-1) and/or the K2-x00 user manual, chapter
@h    "CE conformity, directives and standards".

This AB chekcs if cold drop can be activated.
This is only possible if nozzle moves bwd during autocycle.
An alarm is displayed, if there is no nozzle bwd movement and cold drop is activated.

*)

IMPORT_OVER_LISTFILE
 cCompODC
, tnNozzleBackMode
, tsDeviceId
, tsColdDropParams
, KSYS_Status

END_IMPORT

ALGORITHM_BLOCK ABCheckColdDropPossible #DUMMY_EDIT_BLOCK

SYSTEM_VAR
 sv_DeviceId : tsDeviceId;
 sv_ColdDropSettings : tsColdDropParams;
END_VAR

SYSTEM_OBJECT
 erColdDropNotPossible : ALARM;
 TaskMid : TASK;
 PU_Task_7 : TASK;
END_OBJECT

VAR
 mpNozzleBwdMode : REFTO tnNozzleBackMode;
END_VAR

ALGORITHM aCheck

#BEGIN_EDIT_BLOCK
(**************************************** WARNING ********************************************
 *** The KEBA Kemro K2 System including software is not intended for safety control tasks! ***
 ***                       For further information see Comment tab!                        ***
 *********************************************************************************************)

//cold drop is only possible if nozzle moves bwd during autocycle
IF sv_ColdDropSettings.bUse AND mpNozzleBwdMode^ = nNoNozzleBack THEN
   SET_ALARM(Name := erColdDropNotPossible,
             SubID1 := sv_DeviceId.CompId,
             SubID2 := sv_DeviceId.IndexId);
ELSE
   RESET_ALARM(Name := erColdDropNotPossible,
             SubID1 := sv_DeviceId.CompId,
             SubID2 := sv_DeviceId.IndexId);
END_IF;

;#END_EDIT_BLOCK END_ALGORITHM

POSTUPDATE_ALGORITHM pCheckColdDropPossible ON PU_Task_7 WITH mpNozzleBwdMode^,sv_ColdDropSettings.bUse

#BEGIN_EDIT_BLOCK
(**************************************** WARNING ********************************************
 *** The KEBA Kemro K2 System including software is not intended for safety control tasks! ***
 ***                       For further information see Comment tab!                        ***
 *********************************************************************************************)

aCheck();

;#END_EDIT_BLOCK END_ALGORITHM

PROCESS_ALGORITHM paInit ON TaskMid AUTOSTART

VAR
 Status : KSYS_Status;
 sVarName : STRING(255);
END_VAR
#BEGIN_EDIT_BLOCK
(**************************************** WARNING ********************************************
 *** The KEBA Kemro K2 System including software is not intended for safety control tasks! ***
 ***                       For further information see Comment tab!                        ***
 *********************************************************************************************)

//get refto nozzle back mode (located in Nozzle - fu)
sVarName := CONCAT('Nozzle',DINT_TO_STRING(sv_DeviceId.IndexId),'.sv_NozzleBwdMode');
mpNozzleBwdMode := GET_SYNC_REFTO(sVarName, T#0s, Status);

aCheck();

STOP_PROCESS_ALGORITHM();

;#END_EDIT_BLOCK END_ALGORITHM

END_ALGORITHM_BLOCK

#END_OF_IEC_PART

@Puma @IecEditor 6 97 @Pou 25
@@@BEG_Comment@@@
@h    ! WARNING !
@h    The Kemro K2 system (including software) only meets category B according to EN 954-1,
@h    thus it is not intended for usage in safety-relevant control applications in the field
@h    of personal safety (e.g. emergency stop).
@h    To implement potentially necessary safety-relevant control tasks, always use additional
@h    external safety devices that are intended for the particular purpose, and meet the necessary
@h    functional safety.
@h    For further information see EN 954-1 (EN ISO 13849-1) and/or the K2-x00 user manual, chapter
@h    "CE conformity, directives and standards".

This AB chekcs if cold drop can be activated.
This is only possible if nozzle moves bwd during autocycle.
An alarm is displayed, if there is no nozzle bwd movement and cold drop is activated.

@@@END_Comment@@@

@BEG_Contents

@BEG_Func
@RT(17)FuncTreeContainer
0
@END_Func

@BEG_Const
@RT(18)ConstTreeContainer
1
@Var @RT(8)cCompODC @RT(0) @T @F @DT @RT(4)DINT @RT(0) @T @T @BASIC 0 @F
@F @F
@T
@BEG_Attrib
0 @RT(3)136 @RT(13)Component ODC
@END_Attrib
1 1 @F @F @F @F

@END_Const

@BEG_Export

@BEG_Kind
@ALGORITHM_BLOCK @RT(23)ABCheckColdDropPossible @STRUCTURED_TEXT
@RT(0) @RT(0) @RT(0)
@END_Kind

@BEG_Dcl
@RT(16)DclTreeContainer
6
@Var @RT(15)mpNozzleBwdMode @RT(0) @T @T @REFTO 0 @F @DERIVED 0 @T @T @DT @RT(16)tnNozzleBackMode @RT(0) @T @T @UNKNOWN 0 @F
@F @F
@T
@BEG_Attrib
3 @RT(0) @RT(0) @RT(0)
@END_Attrib
1 0 @F @F @F @F

@Var @RT(21)erColdDropNotPossible @RT(0) @T @F @DT @RT(5)ALARM @RT(0) @T @T @BASIC 0 @F
@F @F
@T
@BEG_Attrib
3 @RT(0) @RT(0) @RT(0)
@END_Attrib
1 7 @F @F @F @F

@Var @RT(7)TaskMid @RT(0) @T @F @DT @RT(4)TASK @RT(0) @T @T @BASIC 0 @F
@F @F
@T
@BEG_Attrib
3 @RT(0) @RT(0) @RT(0)
@END_Attrib
1 7 @F @F @F @F

@Var @RT(9)PU_Task_7 @RT(0) @T @F @DT @RT(4)TASK @RT(0) @T @T @BASIC 0 @F
@F @F
@T
@BEG_Attrib
3 @RT(0) @RT(0) @RT(0)
@END_Attrib
1 7 @F @F @F @F

@Var @RT(11)sv_DeviceId @RT(0) @T @T @DERIVED 0 @T @T @DT @RT(10)tsDeviceId @RT(0) @T @T @UNKNOWN 0 @F
@F @F
@T
@BEG_Attrib
3 @RT(0) @RT(0) @RT(0)
@END_Attrib
1 8 @F @F @F @F

@Var @RT(19)sv_ColdDropSettings @RT(0) @T @T @DERIVED 0 @T @T @DT @RT(16)tsColdDropParams @RT(0) @T @T @UNKNOWN 0 @F
@F @F
@T
@BEG_Attrib
3 @RT(0) @RT(0) @RT(0)
@END_Attrib
1 8 @F @F @F @F

@END_Dcl

@END_Export

@BEG_Body

3

@BEG_Export

@BEG_Algo
@ALGORITHM @RT(6)aCheck @STRUCTURED_TEXT
@RT(0) @RT(0) @RT(0) @F @F
@END_Algo

@BEG_Dcl
@RT(16)DclTreeContainer
0
@END_Dcl

@END_Export

@BEG_Export

@BEG_Algo
@POSTUPDATE_ALGORITHM @RT(22)pCheckColdDropPossible @STRUCTURED_TEXT
@RT(0) @RT(41)mpNozzleBwdMode^,sv_ColdDropSettings.bUse @RT(9)PU_Task_7 @F @F
@END_Algo

@BEG_Dcl
@RT(16)DclTreeContainer
0
@END_Dcl

@END_Export

@BEG_Export

@BEG_Algo
@PROCESS_ALGORITHM @RT(6)paInit @STRUCTURED_TEXT
@RT(0) @RT(0) @RT(7)TaskMid @T @F
@END_Algo

@BEG_Dcl
@RT(16)DclTreeContainer
2
@Var @RT(6)Status @RT(0) @T @T @DERIVED 0 @T @T @DT @RT(11)KSYS_Status @RT(0) @T @T @UNKNOWN 0 @F
@F @F
@T
@BEG_Attrib
3 @RT(0) @RT(0) @RT(0)
@END_Attrib
1 0 @F @F @F @F

@Var @RT(8)sVarName @RT(0) @T @F @DT @RT(11)STRING(255) @RT(0) @T @T @STRING 0 @F @RT(3)255 @F
@F @F
@T
@BEG_Attrib
3 @RT(0) @RT(0) @RT(0)
@END_Attrib
1 0 @F @F @F @F

@END_Dcl

@END_Export

@BEG_Body
@TL(16)
(**************************************** WARNING ********************************************
 *** The KEBA Kemro K2 System including software is not intended for safety control tasks! ***
 ***                       For further information see Comment tab!                        ***
 *********************************************************************************************)

//cold drop is only possible if nozzle moves bwd during autocycle
IF sv_ColdDropSettings.bUse AND mpNozzleBwdMode^ = nNoNozzleBack THEN
   SET_ALARM(Name := erColdDropNotPossible,
             SubID1 := sv_DeviceId.CompId,
             SubID2 := sv_DeviceId.IndexId);
ELSE
   RESET_ALARM(Name := erColdDropNotPossible,
             SubID1 := sv_DeviceId.CompId,
             SubID2 := sv_DeviceId.IndexId);
END_IF;

@END_Body

@@@BEG_Comment@@@
@TL(0)

@@@END_Comment@@@

@BEG_Body
@TL(7)
(**************************************** WARNING ********************************************
 *** The KEBA Kemro K2 System including software is not intended for safety control tasks! ***
 ***                       For further information see Comment tab!                        ***
 *********************************************************************************************)

aCheck();

@END_Body

@@@BEG_Comment@@@
@TL(0)

@@@END_Comment@@@

@BEG_Body
@TL(13)
(**************************************** WARNING ********************************************
 *** The KEBA Kemro K2 System including software is not intended for safety control tasks! ***
 ***                       For further information see Comment tab!                        ***
 *********************************************************************************************)

//get refto nozzle back mode (located in Nozzle - fu)
sVarName := CONCAT('Nozzle',DINT_TO_STRING(sv_DeviceId.IndexId),'.sv_NozzleBwdMode');
mpNozzleBwdMode := GET_SYNC_REFTO(sVarName, T#0s, Status);

aCheck();

STOP_PROCESS_ALGORITHM();

@END_Body

@@@BEG_Comment@@@
@TL(0)

@@@END_Comment@@@
@END_Body

@END_Contents
